(* PLC project simul_visu_rmll, lolitech simul_visu_rmll 1 *)
(* stored: creationDateTime 2008-06-27 17:09:17, modificationDateTime 2008-08-28 16:32:51 *)

TYPE gauge_range : INT(0..100);
END_TYPE

PROGRAM main
  VAR
    pump_in AT %IX2.0.8192.0 : BOOL;
    full_out AT %QX2.0.8194.0 : BOOL;
    empty_out AT %QX2.0.8195.0 : BOOL;
    sink_in AT %IX2.0.8193.0 : BOOL;
    gauge_out AT %QW2.0.8196.0 : gauge_range := 0;
  END_VAR
  VAR
    led_full : Button;
    led_pump : Button;
    led_sink : Button;
    led_empty : Button;
    movewater : Transform;
  END_VAR
  VAR
    tmp1 AT %QD1.0.1 : REAL;
    tmp2 AT %QW1.0.0 : INT;
  END_VAR
  VAR  (* added by the conversion: wires and edge detectors of the diagram *)
    _SUB17_OUT : INT;
    _ADD35_OUT : REAL;
  END_VAR

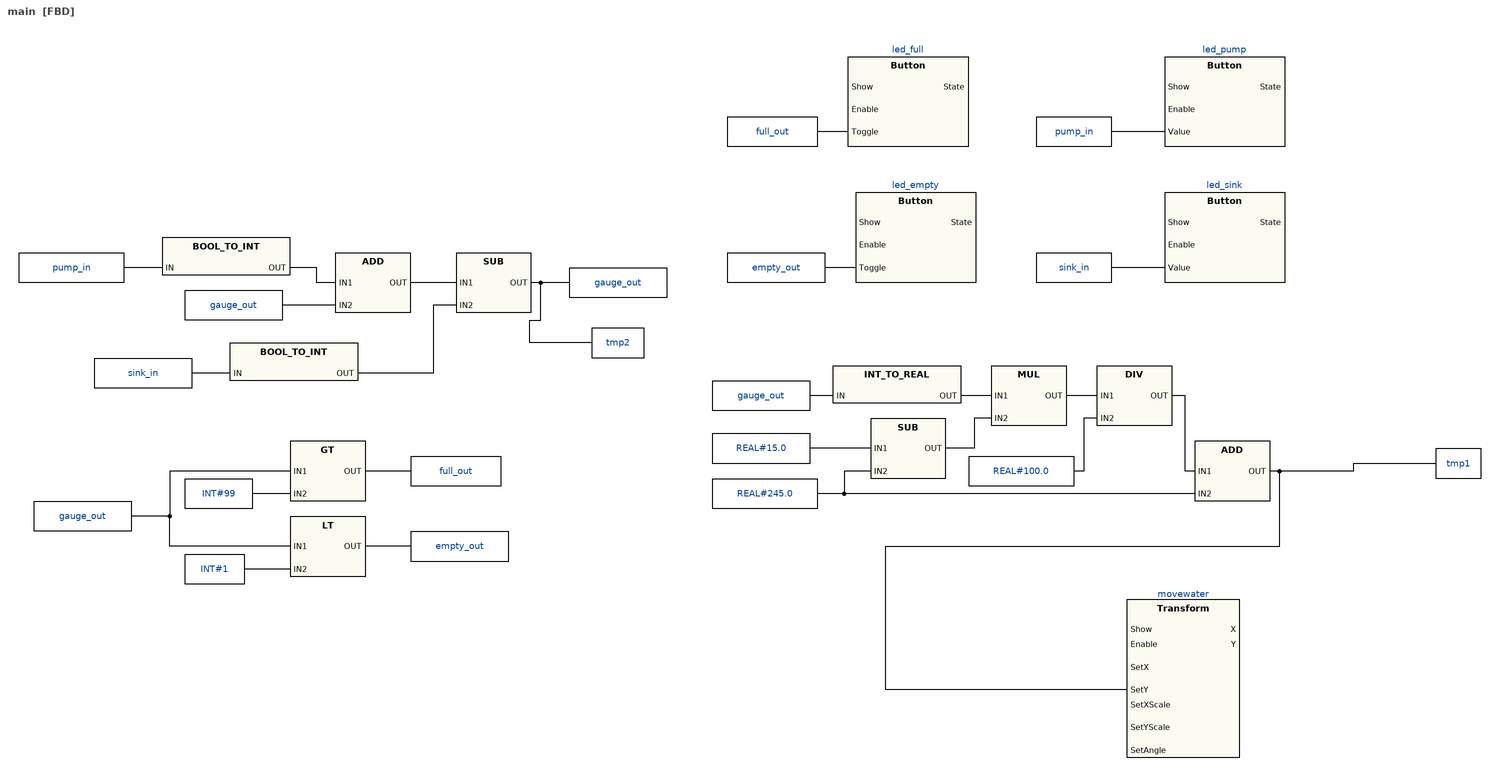
(* FBD diagram, written out as Structured Text *)
_SUB17_OUT := BOOL_TO_INT(pump_in) + gauge_out - BOOL_TO_INT(sink_in);
gauge_out := _SUB17_OUT;
tmp2 := _SUB17_OUT;
full_out := gauge_out > INT#99;
_ADD35_OUT := INT_TO_REAL(gauge_out) * (REAL#15.0 - REAL#245.0) / REAL#100.0 + REAL#245.0;
tmp1 := _ADD35_OUT;
empty_out := gauge_out < INT#1;
led_full(Toggle := full_out);
led_pump(Value := pump_in);
led_empty(Toggle := empty_out);
led_sink(Value := sink_in);
movewater(SetY := _ADD35_OUT);
END_PROGRAM

CONFIGURATION conf
  RESOURCE ress ON PLC
    TASK matache(INTERVAL := 00:00:00.100000, PRIORITY := 0);
    PROGRAM moninst WITH matache : main;
  END_RESOURCE
END_CONFIGURATION
